// Mitsubishi GX Works2 project: IELET2103_Øving3   PLC: FX2N/FX2NC
// IELET2103_Øving3

// global labels: Global1
VAR_GLOBAL
  seq : INT;
  Start AT M100 : BOOL;
  Stopp AT M101 : BOOL;
  Dreieretning AT M102 : BOOL;
  Modulplass0 : INT;
END_VAR

// task Task_01 (event TRUE, interval 0, priority 31): Oppgave3

PROGRAM Oppgave1a)
VAR
  TON_1 : TON;
  tid : WORD;
END_VAR
(* structured ladder/FBD written out as ST: instructions are called as NAME(EN, inputs, outputs); _pN, _eN, _tN stand for wires *)
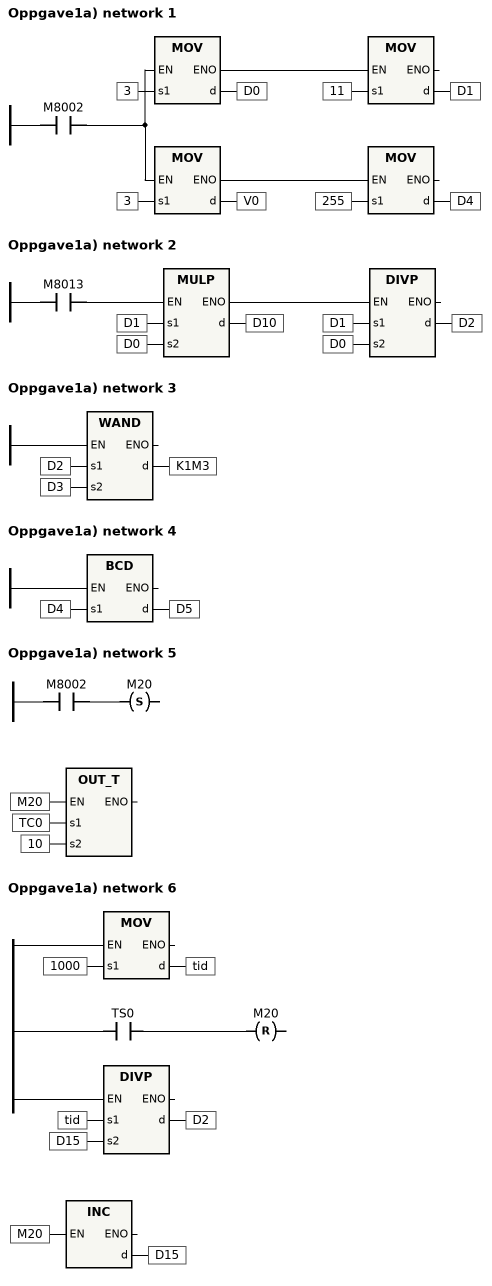
(* network 1 *)
_e1 := MOV(M8002, 3, D0);
MOV(_e1, 11, D1);
_e2 := MOV(M8002, 3, V0);
MOV(_e2, 255, D4);
(* network 2 *)
_e1 := MULP(M8013, D1, D0, D10);
DIVP(_e1, D1, D0, D2);
(* network 3 *)
WAND(TRUE, D2, D3, K1M3);
(* network 4 *)
BCD(TRUE, D4, D5);
(* network 5 *)
SET(M8002, M20);
OUT_T(M20, TC0, 10);
(* network 6 *)
RST(TS0, M20);
INC(M20, D15);
MOV(TRUE, 1000, tid);
DIVP(TRUE, tid, D15, D2);
END_PROGRAM

PROGRAM Oppgave1b)
(* structured ladder/FBD written out as ST: instructions are called as NAME(EN, inputs, outputs); _pN, _eN, _tN stand for wires *)
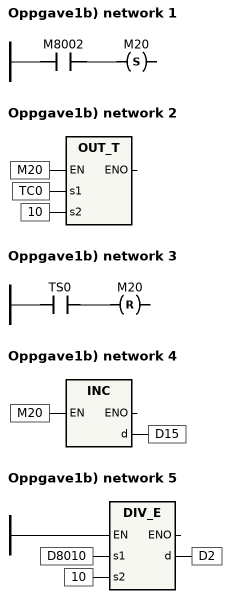
(* network 1 *)
SET(M8002, M20);
(* network 2 *)
OUT_T(M20, TC0, 10);
(* network 3 *)
RST(TS0, M20);
(* network 4 *)
INC(M20, D15);
(* network 5 *)
DIV_E(TRUE, D8010, 10, D2);
END_PROGRAM

PROGRAM Oppgave1c)
(* structured ladder/FBD written out as ST: instructions are called as NAME(EN, inputs, outputs); _pN, _eN, _tN stand for wires *)
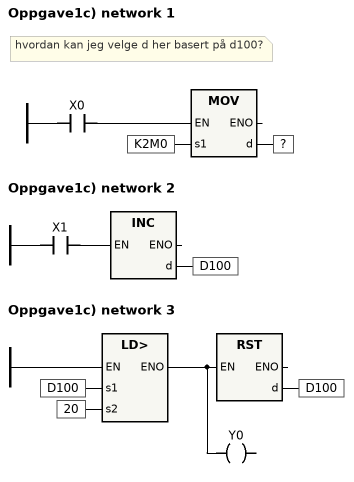
(* network 1 *)
(* hvordan kan jeg velge d her basert på d100? *)
MOV(X0, K2M0, ?);
(* network 2 *)
INC(X1, D100);
(* network 3 *)
_e1 := LD>(TRUE, D100, 20);
Y0 := _e1;
RST(_e1, D100);
END_PROGRAM

PROGRAM Oppgave1d)
(* structured ladder/FBD written out as ST: instructions are called as NAME(EN, inputs, outputs); _pN, _eN, _tN stand for wires *)
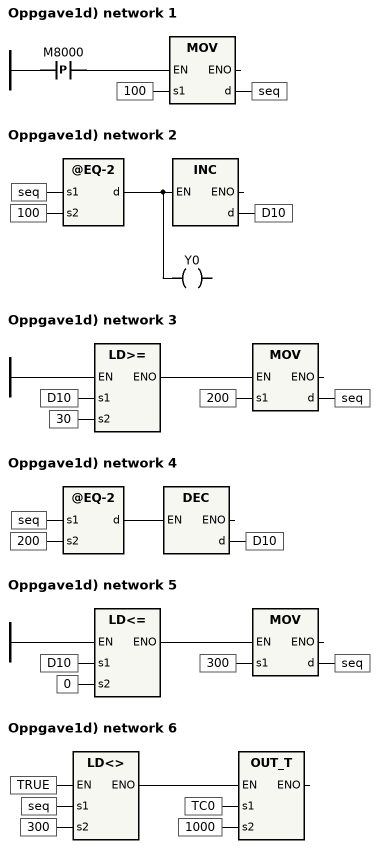
(* network 1 *)
MOV(LDP(TRUE, M8000), 100, seq);
(* network 2 *)
_p1 := @EQ-2(seq, 100);
INC(_p1, D10);
Y0 := _p1;
(* network 3 *)
_e1 := LD>=(TRUE, D10, 30);
MOV(_e1, 200, seq);
(* network 4 *)
DEC(@EQ-2(seq, 200), D10);
(* network 5 *)
_e1 := LD<=(TRUE, D10, 0);
MOV(_e1, 300, seq);
(* network 6 *)
_e1 := LD<>(TRUE, seq, 300);
OUT_T(_e1, TC0, 1000);
END_PROGRAM

PROGRAM Oppgave2
VAR
  D0tmp : INT;
END_VAR
(* structured ladder/FBD written out as ST: instructions are called as NAME(EN, inputs, outputs); _pN, _eN, _tN stand for wires *)
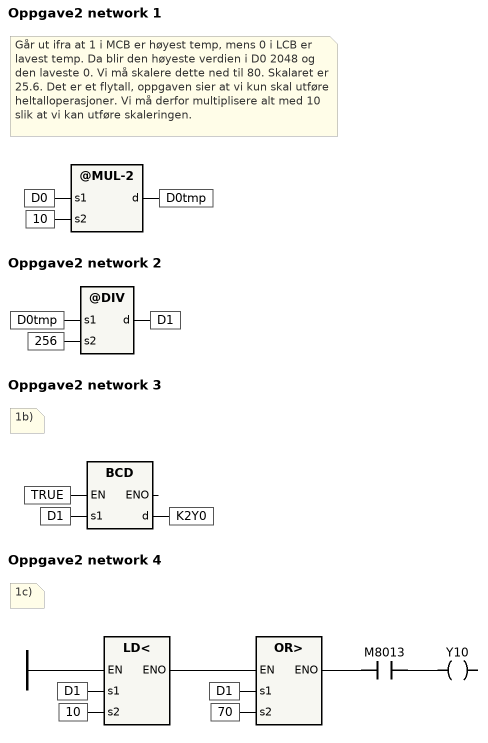
(* network 1 *)
(* Går ut ifra at 1 i MCB er høyest temp, mens 0 i LCB er lavest temp. Da blir den høyeste verdien i D0 2048 og den laveste 0. Vi må skalere dette ned til 80. Skalaret er 25.6. Det er et flytall, oppgaven sier at vi kun skal utføre heltalloperasjoner. Vi må derfor multiplisere alt med 10 slik at vi kan utføre skaleringen. *)
D0tmp := @MUL-2(D0, 10);
(* network 2 *)
D1 := @DIV(D0tmp, 256);
(* network 3 *)
(* 1b) *)
BCD(TRUE, D1, K2Y0);
(* network 4 *)
(* 1c) *)
_e1 := LD<(TRUE, D1, 10);
_e2 := OR>(_e1, D1, 70);
Y10 := _e2 AND M8013;
END_PROGRAM

PROGRAM Oppgave3
VAR
  D100tmp : INT;
  D100DW : DINT;
END_VAR
(* structured ladder/FBD written out as ST: instructions are called as NAME(EN, inputs, outputs); _pN, _eN, _tN stand for wires *)
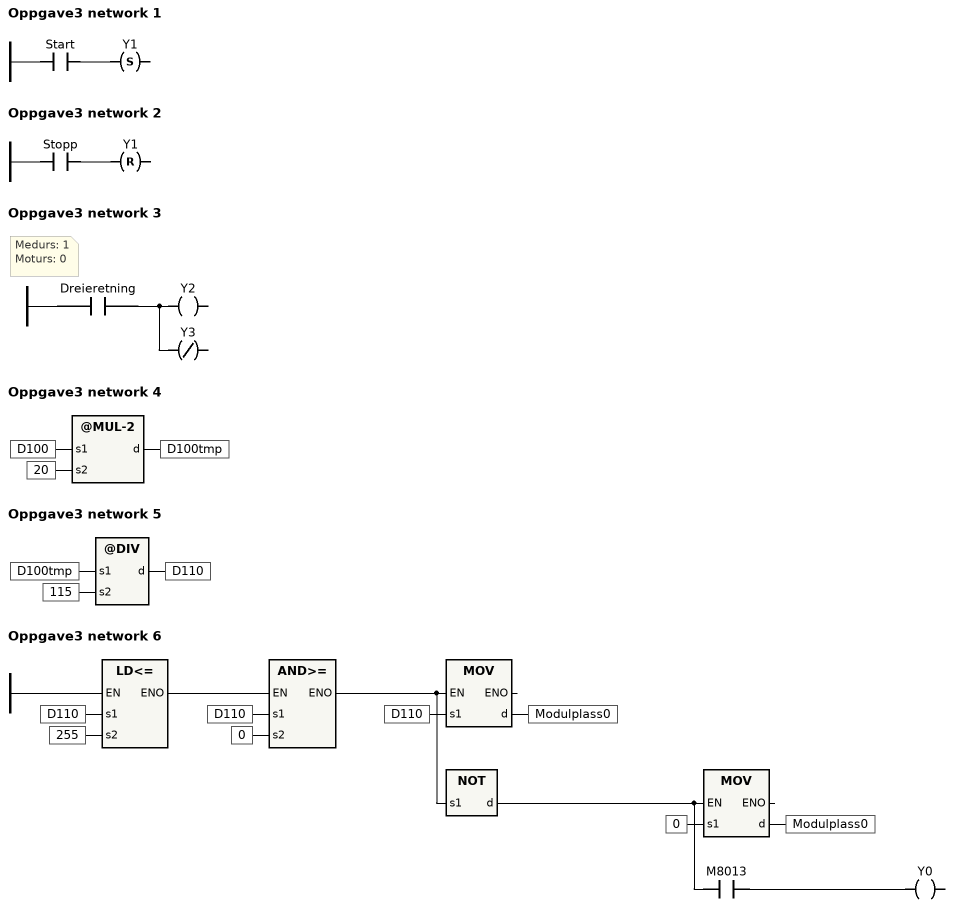
(* network 1 *)
SET(Start, Y1);
(* network 2 *)
RST(Stopp, Y1);
(* network 3 *)
(* Medurs: 1 / Moturs: 0 *)
Y2 := Dreieretning;
Y3 := NOT Dreieretning;
(* network 4 *)
D100tmp := @MUL-2(D100, 20);
(* network 5 *)
D110 := @DIV(D100tmp, 115);
(* network 6 *)
_e1 := LD<=(TRUE, D110, 255);
_e2 := AND>=(_e1, D110, 0);
MOV(_e2, D110, Modulplass0);
_p3 := NOT(_e2);
Y0 := _p3 AND M8013;
MOV(_p3, 0, Modulplass0);
END_PROGRAM
